// TIA Portal V20 export
DATA_BLOCK "FlexNetQuery01"   // DB264
// stored: Access Published, MemoryReserve 100, Namespace PFE
   VAR
      "TraceCode.Data" : String;   // Character String from Host
      Status1 : Array[0..31] of Bool;
   END_VAR
BEGIN
   // Status1[0] : Process 1 Pass/Fail
   // Status1[1] : Process 2 Pass/Fail
   // Status1[2] : Process 3 Pass/Fail
   // Status1[3] : Process 4 Pass/Fail
   // Status1[4] : Process 5 Pass/Fail
   // Status1[5] : Process 6 Pass/Fail
   // Status1[6] : Process 7 Pass/Fail
   // Status1[7] : Process 8 Pass/Fail
   // Status1[8] : Process 9 Pass/Fail
   // Status1[9] : Process 10 Pass/Fail
   // Status1[10] : Process 11 Pass/Fail
   // Status1[30] : New Data
   // Status1[31] : Job Not Found
END_DATA_BLOCK
